Universal Robots URScript: mainUR5.script

def mainUR5():

  #Global Parameters
  global blend_radius_m = 0.001

  #Global parameters  between cam and tcp
  dx = 1.64
  dy = 108.57
  dz = 63.37

  ##############################################################################################################################
  ##############################################################################################################################
  ##################################################### STATES & FUNCTIONS #####################################################
  ##############################################################################################################################
  ##############################################################################################################################

  #######################################################
  ############### FOO_1 SET DESIRED SPEED ###############
  #######################################################

  def set_Speed(vel_ms, vel_rads, acel_ms, acel_rads ):
    #default: speed_ms = 0.3 speed_rads = 0.75 accel_mss = 3 accel_radss = 1.2
    global speed_ms = vel_ms
    global speed_rads = vel_rads
    global accel_mss = acel_ms
    global accel_radss = acel_rads
  end

  #######################################################
  ############# FOO_2 WRITE IN REGISTER INT #############
  #######################################################

  def write_state_int(register, value):
    write_output_integer_register(register, value)
    sleep(0.1)
  end

  #######################################################
  ############# FOO_3 READ IN REGISTER INT ##############
  #######################################################

  def read_state_int(register):
    while (read_input_integer_register(register) ==   -1  ):
      sync()
    end
    return(read_input_integer_register(register))
  end

  #######################################################
  ############# FOO_4 INITIALIZE REGISTER ###############
  #######################################################

  def init_register(register0, register1, register2, value):
    write_state_int(register0, value)
    write_state_int(register1, value)
    write_state_int(register2, value)
  end

  #######################################################
  ################ FOO_5 RESET REGISTER #################
  #######################################################

  def reset_register(register0, register1, register2, value):
    write_state_int(register0, value)
    write_state_int(register1, value)
    write_state_int(register2, value)
    write_state_int(register0, 10)
    write_state_int(register1, 10)
    write_state_int(register2, 10)
  end

  #######################################################
  ############### FOO_6 INITIALIZE STATUS ###############
  #######################################################

  def init_status(register0, register1, register2):
    global status0=read_state_int(register0)
    global status1=read_state_int(register1)
    global status2=read_state_int(register2)
  end

  #######################################################
  ######## FOO_7 CHECK STATUS RECEIVED FROM PLC #########
  #######################################################

	def CheckStatus(state):

	if (status0==state and status1==state and status2==state or status0==state and status1==state and status2!=state or status0==state and status1!=state and
	 status2==state or status0!=state and status1==state and status2==state):
	  return True
	else:
	  return False
	end

	end

  #######################################################
  ############# FOO_8 WRITE IN REGISTER BOOL ############
  #######################################################

	def write_state_bool(register):
	  write_output_boolean_register(register, True)
  	sleep(0.1)
  	write_output_boolean_register(register, False)
	end

<<<<<<< HEAD

=======
  ######################################################################
  #### FOO_9 CHECKS IF THE SEPARATOR HAS BEEN TAKEN BY THE GRIPPER #####
  ######################################################################

	def CheckGripState(number):
		if(gripkit_easy_get_state()==number):
		  return True
		else:
		  return False
		end
	end

  ######################################################################
  ## THREAD_1 MAKE SURE THE GRIPPER IS ALWAYS GRIPPING WHEN IT HAS TO ##
  ######################################################################

  	#thread AlwaysCloseGripper(start):
	  #while(True):
	#	if gripkit_easy_get_state()!=3: #3=gripping
	#		gripkit_easy_grip()
	#	end
	#	sync()
	#  end
  	#end	#use commands: "start_thrd = run AlwaysCloseGripper_thrd()"   and    "kill start_thrd"  IN order to init and stop the thread execution
>>>>>>> f22cb63e4ae80d34c03a3f99a4faca3843d8850d

  ##############################################
  ############### STATE_0 HOMING ###############
  ##############################################

	def UR5Home():

	  init_register(3,4,5,500)
  	#gripkit_easy_enable()  #ESTO DEBERIA IR EN LA MARCHA DE PREPARACIÓN
	  movej([0.000000, -0.174533, -2.775074, -0.349066, 1.570796, 1.570796],accel_radss,speed_rads,0,blend_radius_m)
  	reset_register(3,4,5,501)

	end

  #########################################################################
  ############### STATE_1 PLACE THE CAMERA ON THE FIRST HEAD ##############
  #########################################################################

	def UR5Camera1():

	  init_register(3,4,5,510)
	  movej([0.180484, -1.614237, -2.019210, -1.097497, 1.576100, 3.328193],accel_radss,speed_rads,0,blend_radius_m)
  	movel(p[480.49/1000, -145.25/1000, 239.41/1000, 2.229, 2.216, -0.004], accel_mss, speed_ms, 0, blend_radius_m)
  	reset_register(3,4,5,511)

	end


  ########################################################################
  ####################### STATE_2 GO TO THE BUFFER #######################
  ########################################################################

	def UR5DropHead():

	  init_register(3,4,5,520)
  	movej([-0.064989, -1.480966, -2.238766, -1.013674, 1.573186, 3.082741],accel_radss,speed_rads,0,blend_radius_m)
	  movej([-0.382430, -1.654966, -2.063825, -1.011365, 1.578471, 2.765253],accel_radss,speed_rads,0,blend_radius_m)
<<<<<<< HEAD
  	movel(p[377.91/1000, -384.22/1000, 87.47/1000, 2.238, 2.229, -0.007], accel_mss, speed_ms, 0, blend_radius_m)
=======
  	movel(p[379.05/1000, -370.77/1000, 87.47/1000, 2.219, 2.191, -0.064], accel_mss, speed_ms, 0, blend_radius_m)
>>>>>>> f22cb63e4ae80d34c03a3f99a4faca3843d8850d
  	reset_register(3,4,5,521)

	end

  ###################################################################
  ########## STATE_3 PLACE THE CAMERA ON THE SECOND HEAD  ###########
  ###################################################################

	def UR5Camera2():

  	init_register(3,4,5,530)
<<<<<<< HEAD
=======
    movej(p[377.000/1000, -377.000/1000, 298.000/1000, -2.213, -2.200, 0.000], accel_radss, speed_rads, 0, blend_radius_m)
>>>>>>> f22cb63e4ae80d34c03a3f99a4faca3843d8850d
  	movej([-0.181619, -1.411765, -2.033627, -1.039257, 1.538940, 1.678820],accel_radss,speed_rads,0,blend_radius_m)
  	movej([0.063264, -1.634060, -2.003714, -1.074618, 1.570793, 0.063264],accel_radss,speed_rads,0,blend_radius_m)
  	movel(p[480.49/1000, -9.68/1000, 239.41/1000, 2.239, -2.204, 0], accel_mss, speed_ms, 0, blend_radius_m)
  	reset_register(3,4,5,531)

	end

  ###########################################################################################
  ################ STATE_4 PLACE THE CAMERA ON THE FIRST HEAD TO BE SCREWED  #################
  ###########################################################################################

	def UR5UpCamera1():

  	init_register(3,4,5,540)
  	UR5Home()
  	movej([0.000013, -1.248457, -0.805313, -2.657065, 1.570785, 1.570809],accel_radss,speed_rads,0,blend_radius_m)
<<<<<<< HEAD
  	movej([0.098088, -1.956085, -0.058950, -2.697358, 1.570793, 0.098088],accel_radss,speed_rads,0,blend_radius_m)
  	movel(p[429.86/1000, -10.03/1000, 740.66/1000, 2.206, -2.235, 0.003], accel_mss, speed_ms, 0, blend_radius_m)
=======
  	#movej([0.098088, -1.956085, -0.058950, -2.697358, 1.570793, 0.098088],accel_radss,speed_rads,0,blend_radius_m)
    movej(p[372.000/1000, -8.245/1000, 755.000/1000, 2.221, -2.221, 0.000], accel_radss, speed_rads, 0, blend_radius_m)
  	movel(p[388.0/1000, -8.7/1000, 747.2/1000, 2.279, -2.162, 0.000], accel_mss, speed_ms, 0, blend_radius_m)
>>>>>>> f22cb63e4ae80d34c03a3f99a4faca3843d8850d
  	reset_register(3,4,5,541)

	end

  ###########################################################################################
  ############## STATE_5 GOES DOWN FROM THE SCREWING TO THE BUFFER POSITION  ################
  ###########################################################################################

	def UR5TakeBuffer():

  	init_register(3,4,5,550)
  	movej([0.000013, -1.248457, -0.805313, -2.657065, 1.570785, 1.570809],accel_radss,speed_rads,0,blend_radius_m)
<<<<<<< HEAD
  	movej([-0.000038, -0.831112, -2.092842, -1.579170, 1.570941, 1.570928],accel_radss,speed_rads,0,blend_radius_m)
=======
  	movej(p[230.288/1000, -134.298/1000, 431.619/1000, 0.000, 2.932, 0.000],accel_radss,speed_rads,0,blend_radius_m)
>>>>>>> f22cb63e4ae80d34c03a3f99a4faca3843d8850d
  	UR5DropHead()
  	reset_register(3,4,5,551)

	end

  ###########################################################################################
  ############### STATE_6 PLACE THE CAMERA ON THE SECOND HEAD TO BE SCREWED  ################
  ###########################################################################################

	def UR5UpCamera2():

  	init_register(3,4,5,560)
  	movej([-0.064989, -1.480966, -2.238766, -1.013674, 1.573186, 3.082741],accel_radss,speed_rads,0,blend_radius_m)
  	movej([0.000000, -1.064203, -2.682014, 0.011213, 1.570796, 1.570796],accel_radss,speed_rads,0,blend_radius_m)
<<<<<<< HEAD
  	movej([-0.000038, -0.831112, -2.092842, -1.579170, 1.570941, 1.570928],accel_radss,speed_rads,0,blend_radius_m)
  	movej([0.000013, -1.248457, -0.805313, -2.657065, 1.570785, 1.570809],accel_radss,speed_rads,0,blend_radius_m)
  	movej([0.211928, -1.884634, -0.221391, -2.621276, 1.594272, 3.353305],accel_radss,speed_rads,0,blend_radius_m)
  	movel(p[435.17/1000, -146.59/1000, 741.93/1000, 2.202, 2.240, 0.003], accel_mss, speed_ms, 0, blend_radius_m)
=======
  	movej(p[230.288/1000, -134.298/1000, 431.619/1000, 0.000, 2.932, 0.000],accel_radss,speed_rads,0,blend_radius_m)
  	movej([0.000013, -1.248457, -0.805313, -2.657065, 1.570785, 1.570809],accel_radss,speed_rads,0,blend_radius_m)
  	#movej([0.211928, -1.884634, -0.221391, -2.621276, 1.594272, 3.353305],accel_radss,speed_rads,0,blend_radius_m)
  	#movel(p[435.17/1000, -146.59/1000, 741.93/1000, 2.202, 2.240, 0.003], accel_mss, speed_ms, 0, blend_radius_m)
    movej(p[372.000/1000, -120.763/1000, 749.000/1000, -2.180, -2.217, -0.001], accel_radss, speed_rads, 0, blend_radius_m)
    movel(p[391.44/1000, -128.50/1000, 747.2/1000, 2.210, 2.177, -0.033], accel_mss, speed_ms, 0, blend_radius_m)
>>>>>>> f22cb63e4ae80d34c03a3f99a4faca3843d8850d
  	reset_register(3,4,5,561)

	end

  ###########################################################################################
  ########## STATE_7 FROM THE INSTALLATION AREA IT RETURNS TO HOME. END OF CICLE  ###########
  ###########################################################################################

	def UR5Return():

  	init_register(3,4,5,570)
  	movej([0.000013, -1.248457, -0.805313, -2.657065, 1.570785, 1.570809],accel_radss,speed_rads,0,blend_radius_m)
<<<<<<< HEAD
  	movej([-0.000038, -0.831112, -2.092842, -1.579170, 1.570941, 1.570928],accel_radss,speed_rads,0,blend_radius_m)
=======
    movej(p[230.288/1000, -134.298/1000, 431.619/1000, 0.000, 2.932, 0.000],accel_radss,speed_rads,0,blend_radius_m)
>>>>>>> f22cb63e4ae80d34c03a3f99a4faca3843d8850d
  	movej([0.000000, -1.064203, -2.682014, 0.011213, 1.570796, 1.570796],accel_radss,speed_rads,0,blend_radius_m)
  	UR5Home()
  	reset_register(3,4,5,571)

	end

  #######################################################
  ####### STATE_8 CONTROL TO CENTER CAM OVER NUT ########
  #######################################################

	def CtrCamPos(x_s,y_s):

		init_register(3,4,5,580)

		#dx: direction of tool movement x-axis
		#dy: direction of tool movement x-axis

		center_ok = True
		while(center_ok):

			#wait for the variable script calculated by the vision system
			while (not(read_input_boolean_register(2) ==   True  )):
				sync()
			end

			center_ok =  not  read_input_boolean_register(3)
			cx = read_input_float_register(0) # x-axis deviation
			cy = read_input_float_register(1) # y-axis deviation
			turn_head = read_input_float_register(2) # picth  deviation

			data_vision = p[ x_s*(cx/1000),y_s*(cy/1000),0,0,0,0] # trasform to position variable in base coordinates
			tcp_inst= get_actual_tcp_pose () # get the actual tcp positions.
			pos_calculate = pose_add (tcp_inst, data_vision )
			movel(pos_calculate, accel_mss, speed_ms, 0, blend_radius_m)

			write_state_bool(2) #write finish operation

			sync()
		end
		reset_register(3,4,5,581)

	end

  #######################################################
  ########### STATE_9 MOVE TO NUT AND DOWN ##############
  #######################################################

	def MoveToNut(dx,dy,dz):

		init_register(3,4,5,590)
		#dx,dy,dz, distance between optical cam center and nut center

		tcp_inst = get_actual_tcp_pose()
		tcp_to_optical_center = p[dx/1000,dy/1000,0,0,0,0]
		pos_nut = pose_add(tcp_inst, tcp_to_optical_center)
		movel(pos_nut ,accel_mss, speed_ms, 0, blend_radius_m)

		write_state_bool(2) #write finish movement

		# wait move servomotot with calculate angle of nut
		while (not(read_input_boolean_register(2) ==   True  )):
		  sync()
		end

		#move tcp-tool to inside nut
		tcp_inst = get_actual_tcp_pose()
		tcp_to_nut = p[0,0,dz/1000,0,0,0]
		pos_nut = pose_add (tcp_inst, tcp_to_nut)
		movel(pos_nut, accel_mss, speed_ms, 0, blend_radius_m)

		# close the tool and check if the head is pressed
<<<<<<< HEAD
		set_tool_digital_out(1, True)
		sleep(3.0)
=======
		gripkit_easy_grip()
		var=CheckGripState(3) #check if the tool has gripped the separator correctly
   	while var!=True:
    	gripkit_easy_release()
	    gripkit_easy_grip()
	  	var=CheckGripState(3)
		end
		#sleep(3.0)
>>>>>>> f22cb63e4ae80d34c03a3f99a4faca3843d8850d

		write_state_bool(2) #write finish movement
		reset_register(3,4,5,591)
	end

  #######################################################
  ############ STATE_10 UNSCREW AND UP TOOL #############
  #######################################################

	def UnScrew():
		init_register(3,4,5,5100)

		#Apply force in z axis to up robot
		limits = [0.1, 0.1, 0.15, 0.34, 0.34, 0.34] #limits or move velocity
		frame = [0,0,0,0,0,0] #tool or base frame
		selection = [0, 0, 1, 0, 0, 0] #[x,y,z,x,ry,rz]
		wrench = [0, 0, 1, 0, 0, 0] # force to apply
		type = 2 #kind or force mode
		zero_ftsensor()

		force_mode(frame, selection , wrench, type, limits)

		# wait to servomotor finish to unscrew
		while (not(read_input_boolean_register(2) ==   True  )):
		  sync()
		end

		# kill force mode
		end_force_mode()

		# Up the robot
		tcp_inst = get_actual_tcp_pose()
		up_distance = p[0,0,40/1000,0,0,0]
		pos_up = pose_add (tcp_inst, up_distance)
    set_payload(3.89,[-102/1000,6/1000,-17/1000]) #adjust new weight of the tool
		movel(pos_up, accel_mss, speed_ms, 0, blend_radius_m)

		write_state_bool(2) #write finish movement

		reset_register(3,4,5,5101)
	end

	#######################################################
	############ STATE_11 MOVE TO NUT AND DOWN ############
	#######################################################

	def Screw():
		init_register(3,4,5,5110)

		#Apply force in z axis to down robot
		limits = [0.1, 0.1, 0.15, 0.34, 0.34, 0.34] #limits or move velocity
		frame = [0,0,0,0,0,0] #tool or base frame
		selection = [0, 0, 1, 0, 0, 0] #[x,y,z,x,ry,rz]
		wrench = [0, 0, -5, 0, 0, 0] # force to apply
		type = 2 #kind or force mode
		zero_ftsensor()

		force_mode(frame, selection , wrench, type, limits)

		write_state_bool(2) #write start screw

		# wait to servomotor finish to screw
		while (not(read_input_boolean_register(2) ==   True  )):
		  sync()
		end

		# kill force mode
		end_force_mode()


		reset_register(3,4,5,5111)
	end

	#######################################################
	########## STATE_12 UP ROBOT AFTER TO SCREW ###########
	#######################################################
	def UpRobotAs():

		init_register(3,4,5,5120)

    #Open the tool
    gripkit_easy_release()
		var=CheckGripState(1) #check if the tool is open
   	while var!=True:
	    gripkit_easy_release()
	  	var=CheckGripState(1)
		end

		#Apply force in z axis to up robot
		limits = [0.1, 0.1, 0.15, 0.34, 0.34, 0.34] #limits or move velocity
		frame = [0,0,0,0,0,0] #tool or base frame
		selection = [0, 0, 1, 0, 0, 0] #[x,y,z,x,ry,rz]
		wrench = [0, 0, 20, 0, 0, 0] # force to apply
		type = 2 #kind or force mode
		zero_ftsensor()

		force_mode(frame, selection , wrench, type, limits)

		# Up the robot
		tcp_inst = get_actual_tcp_pose()
		up_distance = p[0,0,40/1000,0,0,0]
		pos_up = pose_add (tcp_inst, up_distance)
    #set_payload(,[,,]) #back to normal tool weight
		movel(pos_up, accel_mss, speed_ms, 0, blend_radius_m)

		# kill force mode
		end_force_mode()

		write_state_bool(2) #write finish movement

		reset_register(3,4,5,5121)

	end


  ##############################################################################################################################
  ##############################################################################################################################
  ##################################################### MAIN PROGRAMME #########################################################
  ##############################################################################################################################
  ##############################################################################################################################

  set_tcp(p[-0.082500, -0.001000, 0.071500, 0.000000, 0.000000, 0.000000])
  #set_payload(,[,,])
  #set_Speed(0.3, 0.75, 3, 1.2)
  #vel_ms, vel_rads, acel_ms, acel_rads

  #State-Machine
  while(True):
    init_status(0,1,2)

   if (CheckStatus(50)==True):
    set_Speed(0.1, 0.75, 3, 1.2)
    UR5Home()
   elif (CheckStatus(51)==True):
    set_Speed(0.1, 0.75, 3, 1.2)
    UR5Camera1()
   elif (CheckStatus(52)==True):
    set_Speed(0.1, 0.75, 3, 1.2)
    UR5DropHead()
   elif (CheckStatus(53)==True):
    set_Speed(0.1, 0.75, 3, 1.2)
    UR5Camera2()
   elif (CheckStatus(54)==True):
    set_Speed(0.1, 0.75, 3, 1.2)
    UR5UpCamera1()
   elif (CheckStatus(55)==True):
    set_Speed(0.1, 0.75, 3, 1.2)
    UR5TakeBuffer()
   elif (CheckStatus(56)==True):
    set_Speed(0.1, 0.75, 3, 1.2)
    UR5UpCamera2()
   elif (CheckStatus(57)==True):
    set_Speed(0.1, 0.75, 3, 1.2)
    UR5Return()

   elif (CheckStatus(58)==True or CheckStatus(64)==True):
    set_Speed(0.1, 0.75, 3, 1.2)
    CtrCamPos(-1,-1) #58==Camera1 position & 64==UpCamera2 position
   elif (CheckStatus(59)==True or CheckStatus(61)==True or CheckStatus(63)==True or CheckStatus(65)==True ): #59==Camera1 position  61==Camera2 position
    set_Speed(0.1, 0.75, 3, 1.2)                                                                             #63==UpCamera1 position 65==UpCamera2 position
    MoveToNut(dx,dy,dz)
   elif (CheckStatus(60)==True or CheckStatus(62)==True ):
    set_Speed(0.1, 0.75, 3, 1.2)
    CtrCamPos(1,1) #60==Camera2 position & 62==UpCamera1 position

   elif (CheckStatus(66)==True):
    set_Speed(0.1, 0.75, 3, 1.2)
    UnScrew()
   elif (CheckStatus(67)==True):
    set_Speed(0.1, 0.75, 3, 1.2)
    Screw()
   elif (CheckStatus(68)==True):
    set_Speed(0.1, 0.75, 3, 1.2)
    UpRobotAs()
   end
  end
end
